// TIA Portal V17 export
// export: Created 2023-06-23T18:33:36.8847413Z, ExportSetting WithDefaults, DisplayName Totally Integrated Automation Portal, DisplayVersion V17, DisplayName TIA Portal Openness, DisplayVersion V17, DisplayName TIA Portal Version Control Interface, DisplayVersion V17, DisplayName STEP 7 Professional, DisplayVersion V17, DisplayName STEP 7 Safety, DisplayVersion V17, DisplayName WinCC Advanced / Unified PC, DisplayVersion V17
VAR_GLOBAL   // PLC tag table "01_EL-1"
   "iEL-1" AT %I0.4 : Bool;
   "oEL-1s" AT %Q17.6 : Bool;
   "oEL-1f" AT %Q17.7 : Bool;
END_VAR
